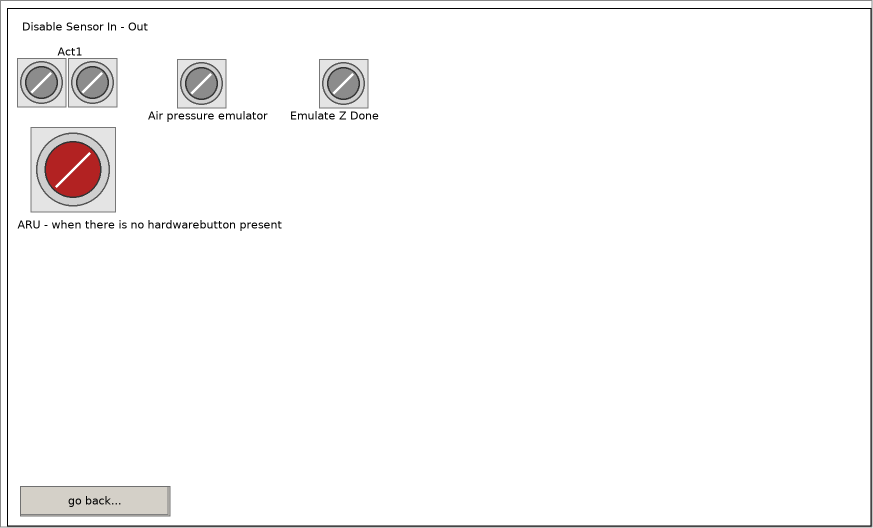
VISUALIZATION VisuAdmin  // 873x528
    Group (265,213 240x84)
        Label (0,0 237x66), "You are not allowed to see this page"
        Label (3,18 237x66), "Please login as another user"
    Rectangle (7,8 864x518)
    Button (20,486 150x30), "go back..."
        OnMouseClick: change screen: Visualization
    Label (-5,37 150x30), "Act1"
    Label (10,12 150x30), "Disable Sensor In - Out"
    RotarySwitch (17,57 49x51), variable: fbAct1.stParam.xPresenceSensIn, behaviour: TOGGLE, style: Switch-RotarySwitch-Gray
    RotarySwitch (68,57 49x51), variable: fbAct1.stParam.xPresenceSensOut, behaviour: TOGGLE, style: Switch-RotarySwitch-Gray
    RotarySwitch (22,127 102x85), variable: stIO.stIn.IxAruIO, behaviour: TOGGLE, style: Switch-RotarySwitch-Red
    Label (1,210 298x30), "ARU - when there is no hardwarebutton present"
    RotarySwitch (177,58 49x51), variable: stio.stIn.xAirPressureOk, behaviour: TOGGLE, style: Switch-RotarySwitch-Gray
    Label (145,101 298x30), "Air pressure emulator"
    Label (287,101 298x30), "Emulate Z Done"
    RotarySwitch (319,58 49x51), variable: stIO.stIn.xEmulateZDone, behaviour: TOGGLE, style: Switch-RotarySwitch-Gray
END_VISUALIZATION

(* stored: Version 1.1.0.1, ProductVersion 3.1.4020.12
   Visu VisuAdmin: Id {6b6a12a9-332a-46cc-9275-7970492bc41a} *)
